PROGRAM MAIN
VAR
	
	
END_VAR


//fbSiemensCameraMV5xCtrl();

//PRG_Test();
PRG_ButtonsHandler();

//IO_logic();

PRG_HikrobotHandler();

	
//Outer_IN_Case_Duplicat();

END_PROGRAM

(* stored: Version 1.1.0.1
   POU MAIN: Id {57de771e-4346-4079-9379-3645d39749ca}, SpecialFunc None *)
